// TIA Portal V20 export
// export: Created 2025-12-01T14:56:16.7687931Z, ExportSetting None, DisplayName Totally Integrated Automation Portal, DisplayVersion V20 Update 3, DisplayName TIA Portal Openness, DisplayVersion V20 Update 3, DisplayName TIA Portal Version Control Interface, DisplayVersion V20 Update 3, DisplayName STEP 7 Professional, DisplayVersion V20 Update 3, DisplayName STEP 7 Safety, DisplayVersion V20 Update 2, DisplayName WinCC Basic/Comfort/Advanced, DisplayVersion V20 Update 3, DisplayName WinCC Professional, DisplayVersion V20 Update 3, DisplayName WinCC Unified, DisplayVersion V20 Update 3
TYPE "UDT_Interlock_Etiquetadora_ZETES"
   STRUCT
      In_PowerOn : Bool;   // Entrada etiquetadora en tensión
      In_Online : Bool;   // Entrada etiquetadora online
      In_Consumible : Bool;   // Entrada etiquetadora estado consumible
      In_Bypass : Bool;   // Entrada etiquetadora estado bypass
      In_BrazoRecogido : Bool;   // Entrada etiquetadora brazo recogido
      In_DataReady : Bool;   // Entrada etiquetadora con datos
      In_FinCiclo : Bool;   // Entrada etiquetadora fin de ciclo
      "Byte0.bit7" : Bool;
      Out_InicioCiclo : Bool;   // Salida etiquetadora activar inicio de ciclo
      Byte1_bit1 : Bool;
      Byte1_bit2 : Bool;
      Byte1_bit3 : Bool;
      Byte1_bit4 : Bool;
      Byte1_bit5 : Bool;
      Byte1_bit6 : Bool;
      Byte1_bit7 : Bool;
      Byte2_bit0 : Bool;
      Byte2_bit1 : Bool;
      Byte2_bit2 : Bool;
      Byte2_bit3 : Bool;
      Byte2_bit4 : Bool;
      Byte2_bit5 : Bool;
      Byte2_bit6 : Bool;
      Byte2_bit7 : Bool;
      Byte3_bit0 : Bool;
      Byte3_bit1 : Bool;
      Byte3_bit2 : Bool;
      Byte3_bit3 : Bool;
      Byte3_bit4 : Bool;
      Byte3_bit5 : Bool;
      Byte3_bit6 : Bool;
      Byte3_bit7 : Bool;
   END_STRUCT;
END_TYPE
